(* IEC 61131-3 sources: stc/tests/twincat_dialect, 7 files *)

(* ---- bit_access_test.st ---- *)
(* TwinCAT dialect: bit access on integer and bit-string values.
   `w.n` reads or writes bit n of an ANY_BIT/ANY_INT value. The GVL below is
   named after this file and is not qualified_only, so ECT and Modbus are
   reachable bare. ECT mirrors an EtherCAT image: a struct member holding a
   WORD of packed digital inputs.
*)

TYPE ST_Terminal :
STRUCT
    q_wDigitalInputs : WORD;
END_STRUCT
END_TYPE

TYPE ST_Ect :
STRUCT
    X : ST_Terminal;
END_STRUCT
END_TYPE

TYPE ST_Modbus :
STRUCT
    arr : ARRAY[0..3] OF WORD;
END_STRUCT
END_TYPE

VAR_GLOBAL CONSTANT
    BIT_READY : DINT := 2;
END_VAR

VAR_GLOBAL
    ECT    : ST_Ect;
    Modbus : ST_Modbus;
END_VAR

TEST_CASE 'Bit read on a nested struct member'
    ECT.X.q_wDigitalInputs := 16#0005;
    ASSERT_TRUE(ECT.X.q_wDigitalInputs.0);
    ASSERT_FALSE(ECT.X.q_wDigitalInputs.1);
    ASSERT_TRUE(ECT.X.q_wDigitalInputs.2);
    ASSERT_FALSE(ECT.X.q_wDigitalInputs.15);
END_TEST_CASE

TEST_CASE 'Bit write on an array element sets exactly that bit'
    Modbus.arr[0].3 := TRUE;
    ASSERT_EQ(Modbus.arr[0], 16#0008);
    ASSERT_TRUE(Modbus.arr[0].3);
    ASSERT_FALSE(Modbus.arr[0].2);
    ASSERT_EQ(Modbus.arr[1], 0);
    Modbus.arr[0].3 := FALSE;
    ASSERT_EQ(Modbus.arr[0], 0);
END_TEST_CASE

TEST_CASE 'BYTE, DWORD and LWORD bit writes'
VAR
    b  : BYTE;
    dw : DWORD;
    lw : LWORD;
END_VAR
    b.7 := TRUE;
    ASSERT_EQ(b, 16#80);
    dw.31 := TRUE;
    dw.0 := TRUE;
    ASSERT_EQ(dw, 16#80000001);
    lw.63 := TRUE;
    ASSERT_TRUE(lw.63);
    ASSERT_FALSE(lw.62);
    lw.63 := FALSE;
    ASSERT_EQ(lw, 0);
END_TEST_CASE

TEST_CASE 'Bit index given by a constant'
VAR
    w : WORD;
END_VAR
    w.BIT_READY := TRUE;
    ASSERT_EQ(w, 16#0004);
    ASSERT_TRUE(w.BIT_READY);
END_TEST_CASE

(* ---- enum_test.st ---- *)
(* TwinCAT dialect: enumerations.
   E_Mode is qualified_only, strict and to_string with an explicit UINT base
   type. E_State uses implicit numbering: a value without an initialiser is
   the previous value plus one. E_Plain has neither attribute, so its values
   are reachable bare and TO_STRING gives the number.
*)

{attribute 'qualified_only'}
{attribute 'strict'}
{attribute 'to_string'}
TYPE E_Mode : (a := 0, b := 1, c := 2) UINT;
END_TYPE

TYPE E_State : (tun := 0, rdy := 2, nst);
END_TYPE

TYPE E_Plain : (p0, p1, p2, p3, p4);
END_TYPE

FUNCTION F_Classify : DINT
VAR_INPUT
    m : E_Mode;
END_VAR
    CASE m OF
        E_Mode.a:
            F_Classify := 10;
        E_Mode.b, E_Mode.c:
            F_Classify := 20;
    ELSE
        F_Classify := -1;
    END_CASE
END_FUNCTION

FUNCTION F_Band : DINT
VAR_INPUT
    p : E_Plain;
END_VAR
    CASE p OF
        p0:
            F_Band := 0;
        p1..p3:
            F_Band := 1;
    ELSE
        F_Band := 2;
    END_CASE
END_FUNCTION

TEST_CASE 'CASE with qualified labels'
    ASSERT_EQ(F_Classify(E_Mode.a), 10);
    ASSERT_EQ(F_Classify(E_Mode.b), 20);
    ASSERT_EQ(F_Classify(E_Mode.c), 20);
END_TEST_CASE

TEST_CASE 'CASE with a range label'
    ASSERT_EQ(F_Band(p0), 0);
    ASSERT_EQ(F_Band(p1), 1);
    ASSERT_EQ(F_Band(p3), 1);
    ASSERT_EQ(F_Band(p4), 2);
END_TEST_CASE

TEST_CASE 'Implicit numbering continues from the previous value'
VAR
    s : E_State;
END_VAR
    s := E_State.nst;
    ASSERT_EQ(TO_DINT(s), 3);
    s := rdy;
    ASSERT_EQ(TO_DINT(s), 2);
    ASSERT_EQ(TO_DINT(E_State.tun), 0);
END_TEST_CASE

TEST_CASE 'TO_STRING gives the name for a to_string enum'
VAR
    m : E_Mode;
END_VAR
    m := E_Mode.b;
    ASSERT_EQ(TO_STRING(m), 'b');
END_TEST_CASE

TEST_CASE 'TO_STRING gives the number for a plain enum'
VAR
    p : E_Plain;
END_VAR
    p := p2;
    ASSERT_EQ(TO_STRING(p), '2');
END_TEST_CASE

TEST_CASE 'Inline enum in a VAR block'
VAR
    light : (red, amber, green) := amber;
END_VAR
    ASSERT_TRUE(light = amber);
    light := green;
    ASSERT_TRUE(light = green);
    ASSERT_FALSE(light = red);
END_TEST_CASE

(* ---- named_args_test.st ---- *)
(* TwinCAT dialect: named arguments in FUNCTION calls used as expressions.
   Inputs may be passed by name in any order, mixed with leading positional
   arguments, or omitted to take their declared default. `=>` binds a
   FUNCTION's VAR_OUTPUT, and TwinCAT allows a trailing comma.
*)

FUNCTION F_X : DINT
VAR_INPUT
    a : DINT;
    b : DINT;
END_VAR
    F_X := a * 10 + b;
END_FUNCTION

FUNCTION F_Scale : DINT
VAR_INPUT
    x : DINT;
    step : DINT := 3;
END_VAR
    F_Scale := x * step;
END_FUNCTION

FUNCTION F_DivMod : DINT
VAR_INPUT
    num : DINT;
    den : DINT;
END_VAR
VAR_OUTPUT
    rest : DINT;
END_VAR
    rest := num MOD den;
    F_DivMod := num / den;
END_FUNCTION

TEST_CASE 'Named arguments equal positional ones'
VAR
    n : DINT;
    m : DINT;
END_VAR
    n := F_X(a := 1, b := 2);
    m := F_X(1, 2);
    ASSERT_EQ(n, 12);
    ASSERT_EQ(n, m);
END_TEST_CASE

TEST_CASE 'Named arguments in a different order'
VAR
    n : DINT;
END_VAR
    n := F_X(b := 2, a := 1);
    ASSERT_EQ(n, 12);
END_TEST_CASE

TEST_CASE 'Positional then named arguments'
VAR
    n : DINT;
END_VAR
    n := F_X(4, b := 5);
    ASSERT_EQ(n, 45);
END_TEST_CASE

TEST_CASE 'Omitted input takes its default'
VAR
    n : DINT;
END_VAR
    n := F_Scale(x := 7);
    ASSERT_EQ(n, 21);
    n := F_Scale(x := 7, step := 2);
    ASSERT_EQ(n, 14);
END_TEST_CASE

TEST_CASE 'Output binding on a FUNCTION'
VAR
    q : DINT;
    r : DINT;
END_VAR
    q := F_DivMod(num := 17, den := 5, rest => r);
    ASSERT_EQ(q, 3);
    ASSERT_EQ(r, 2);
END_TEST_CASE

TEST_CASE 'Trailing comma in a call'
VAR
    n : DINT;
END_VAR
    n := F_X(a := 2, b := 3,);
    ASSERT_EQ(n, 23);
END_TEST_CASE

(* ---- action_test.st ---- *)
(* TwinCAT dialect: ACTIONs on a FUNCTION_BLOCK.
   A_Step is declared inside the FB, A_Reset after END_FUNCTION_BLOCK; both
   belong to FB_Counter and run against the instance's own variables, whether
   the FB body calls them or a caller writes inst.A_Step().
*)

FUNCTION_BLOCK FB_Counter
VAR_INPUT
    step : INT;
END_VAR
VAR_OUTPUT
    n : INT;
    edges : INT;
END_VAR
VAR
    edge : R_TRIG;
    pulse : BOOL;
END_VAR
    A_Step();

ACTION A_Step
    n := n + step;
    edge(CLK := pulse);
    IF edge.Q THEN
        edges := edges + 1;
    END_IF
END_ACTION
END_FUNCTION_BLOCK

ACTION A_Reset
    n := 0;
END_ACTION

TEST_CASE 'FB body runs its action on every call'
VAR
    c : FB_Counter;
END_VAR
    c(step := 2);
    c(step := 2);
    ASSERT_EQ(c.n, 4);
END_TEST_CASE

TEST_CASE 'External call to an action declared after the FB'
VAR
    c : FB_Counter;
END_VAR
    c(step := 3);
    ASSERT_EQ(c.n, 3);
    c.A_Reset();
    ASSERT_EQ(c.n, 0);
END_TEST_CASE

TEST_CASE 'External call to an action declared inside the FB'
VAR
    c : FB_Counter;
END_VAR
    c(step := 5);
    c.A_Step();
    ASSERT_EQ(c.n, 10);
END_TEST_CASE

TEST_CASE 'R_TRIG inside an action keeps state across calls'
VAR
    c : FB_Counter;
END_VAR
    c.pulse := TRUE;
    c(step := 1);
    c(step := 1);
    ASSERT_EQ(c.edges, 1);
    c.pulse := FALSE;
    c(step := 1);
    c.pulse := TRUE;
    c(step := 1);
    ASSERT_EQ(c.edges, 2);
    ASSERT_EQ(c.n, 4);
END_TEST_CASE

(* ---- gvl_test.st ---- *)
(* TwinCAT dialect: global variable lists (GVLs).
   The top-level VAR_GLOBAL block below is a GVL named after this file,
   gvl_test. It has no qualified_only attribute, so its variables are
   reachable both as gvl_test.x and as bare x. Every TEST_CASE starts from
   a freshly initialised GVL.
*)

TYPE ST_Pos :
STRUCT
    x : INT;
    y : INT;
END_STRUCT
END_TYPE

VAR_GLOBAL
    counter : INT := 0;
    limit   : INT := 10;
    pos     : ST_Pos;
END_VAR

FUNCTION_BLOCK FB_Counter
VAR_INPUT
    step : INT;
END_VAR
    gvl_test.counter := gvl_test.counter + step;
END_FUNCTION_BLOCK

TEST_CASE 'Qualified read and write'
    ASSERT_EQ(gvl_test.limit, 10);
    gvl_test.counter := gvl_test.counter + 3;
    ASSERT_EQ(gvl_test.counter, 3);
END_TEST_CASE

TEST_CASE 'Unqualified read and write'
    counter := counter + limit;
    ASSERT_EQ(counter, 10);
    ASSERT_EQ(gvl_test.counter, 10);
END_TEST_CASE

TEST_CASE 'Nested struct member write'
    gvl_test.pos.x := 5;
    pos.y := 7;
    ASSERT_EQ(gvl_test.pos.x, 5);
    ASSERT_EQ(gvl_test.pos.y, 7);
END_TEST_CASE

TEST_CASE 'Each test case gets a fresh GVL'
    ASSERT_EQ(counter, 0);
    ASSERT_EQ(gvl_test.pos.x, 0);
END_TEST_CASE

TEST_CASE 'FB body writes the GVL'
VAR
    fbCount : FB_Counter;
END_VAR
    fbCount(step := 2);
    fbCount(step := 2);
    ASSERT_EQ(gvl_test.counter, 4);
END_TEST_CASE

TEST_CASE 'Local variable shadows a GVL variable'
VAR
    limit : INT := 99;
END_VAR
    ASSERT_EQ(limit, 99);
    ASSERT_EQ(gvl_test.limit, 10);
END_TEST_CASE

(* ---- ref_this_super_test.st ---- *)
(* TwinCAT dialect: REF= references, THIS^ and SUPER^.
   `r REF= x;` binds a REFERENCE TO variable to x; reads and writes of r then
   go through to x. Inside a FUNCTION_BLOCK, THIS^ is the current instance
   and an unqualified call to one of its METHODs dispatches on it. In a
   derived FB, SUPER^.M() calls the base implementation and SUPER^() runs
   the base body.
*)

TYPE ST_Pair :
STRUCT
    m : DINT;
    k : DINT;
END_STRUCT
END_TYPE

FUNCTION_BLOCK FB_Base
VAR_OUTPUT
    x : DINT;
    bodyRuns : DINT;
END_VAR
    bodyRuns := bodyRuns + 1;

METHOD Inc : DINT
VAR_INPUT
    step : DINT;
END_VAR
    THIS^.x := THIS^.x + step;
    Inc := THIS^.x;
END_METHOD

METHOD M : DINT
    M := 100;
END_METHOD

METHOD Twice : DINT
    Inc(step := 1);
    THIS^.Inc(step := 1);
    Twice := x;
END_METHOD
END_FUNCTION_BLOCK

FUNCTION_BLOCK FB_Derived EXTENDS FB_Base
VAR_OUTPUT
    fromSuper : DINT;
END_VAR
    SUPER^();
    fromSuper := SUPER^.M();

METHOD M : DINT
    M := SUPER^.M() + 1;
END_METHOD
END_FUNCTION_BLOCK

TEST_CASE 'Reference to a variable reads and writes through'
VAR
    n : DINT;
    r : REFERENCE TO DINT;
END_VAR
    n := 4;
    r REF= n;
    ASSERT_EQ(r, 4);
    r := 9;
    ASSERT_EQ(n, 9);
    n := 11;
    ASSERT_EQ(r, 11);
END_TEST_CASE

TEST_CASE 'Reference to a struct member'
VAR
    s : ST_Pair;
    r : REFERENCE TO DINT;
END_VAR
    r REF= s.m;
    r := 5;
    ASSERT_EQ(s.m, 5);
    ASSERT_EQ(s.k, 0);
END_TEST_CASE

TEST_CASE 'Reference to an array element keeps its element'
VAR
    arr : ARRAY[0..3] OF DINT;
    i : DINT;
    r : REFERENCE TO DINT;
END_VAR
    i := 1;
    r REF= arr[i];
    i := 2;
    r := 7;
    ASSERT_EQ(arr[1], 7);
    ASSERT_EQ(arr[2], 0);
END_TEST_CASE

TEST_CASE 'THIS^ member access and method calls'
VAR
    fb : FB_Base;
    v : DINT;
END_VAR
    v := fb.Inc(step := 3);
    ASSERT_EQ(v, 3);
    ASSERT_EQ(fb.x, 3);
    v := fb.Twice();
    ASSERT_EQ(v, 5);
    ASSERT_EQ(fb.x, 5);
END_TEST_CASE

TEST_CASE 'SUPER^ method call and base body'
VAR
    d : FB_Derived;
END_VAR
    d();
    ASSERT_EQ(d.fromSuper, 100);
    ASSERT_EQ(d.bodyRuns, 1);
    ASSERT_EQ(d.M(), 101);
    d();
    ASSERT_EQ(d.bodyRuns, 2);
END_TEST_CASE

(* ---- empty_args_test.st ---- *)
(* TwinCAT dialect: empty formal arguments.
   TwinCAT writes unused outputs of a call as "Q => ," and treats them as
   omitted. t1 is called with empty output bindings and t2 without them; both
   timers must behave identically.
*)

TEST_CASE 'Empty output bindings run like omitted ones'
VAR
    t1 : TON;
    t2 : TON;
    i : INT;
END_VAR
    FOR i := 1 TO 5 DO
        t1(IN := TRUE, PT := T#100MS, Q => , ET => );
        t2(IN := TRUE, PT := T#100MS);
        ADVANCE_TIME(T#10MS);
    END_FOR
    (* 50 ms elapsed *)
    t1(IN := TRUE, PT := T#100MS, Q => , ET => );
    t2(IN := TRUE, PT := T#100MS);
    ASSERT_FALSE(t1.Q);
    ASSERT_EQ(t1.Q, t2.Q);
    ASSERT_EQ(t1.ET, t2.ET);
    ASSERT_EQ(t1.ET, T#50MS);
END_TEST_CASE

TEST_CASE 'Empty bindings still let the timer elapse'
VAR
    t1 : TON;
    t2 : TON;
    i : INT;
END_VAR
    FOR i := 1 TO 15 DO
        t1(IN := TRUE, PT := T#100MS, Q => , ET => );
        t2(IN := TRUE, PT := T#100MS);
        ADVANCE_TIME(T#10MS);
    END_FOR
    (* 150 ms elapsed *)
    t1(IN := TRUE, PT := T#100MS, Q => , ET => );
    t2(IN := TRUE, PT := T#100MS);
    ASSERT_TRUE(t1.Q);
    ASSERT_EQ(t1.Q, t2.Q);
    ASSERT_EQ(t1.ET, t2.ET);
END_TEST_CASE
